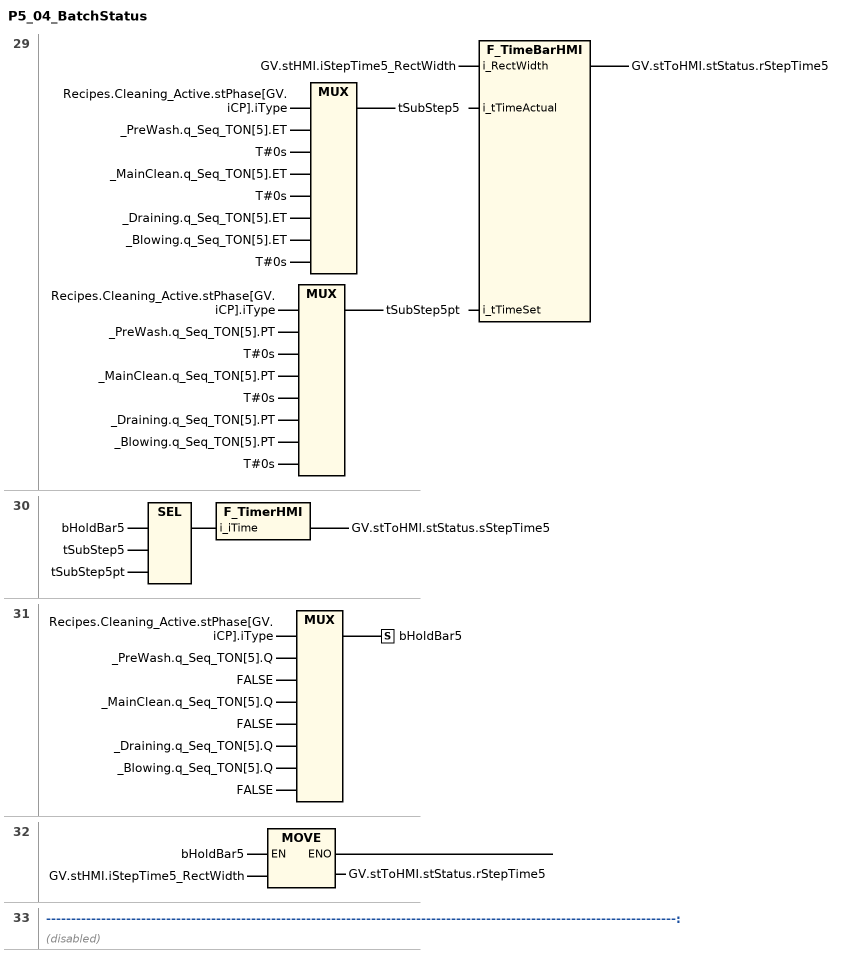
// NETWORK 29
_w10 := MUX(Recipes.Cleaning_Active.stPhase[GV.iCP].iType, _PreWash.q_Seq_TON[5].ET, T#0s, _MainClean.q_Seq_TON[5].ET, T#0s, _Draining.q_Seq_TON[5].ET, _Blowing.q_Seq_TON[5].ET, T#0s);
tSubStep5 := _w10;
_w11 := MUX(Recipes.Cleaning_Active.stPhase[GV.iCP].iType, _PreWash.q_Seq_TON[5].PT, T#0s, _MainClean.q_Seq_TON[5].PT, T#0s, _Draining.q_Seq_TON[5].PT, _Blowing.q_Seq_TON[5].PT, T#0s);
tSubStep5pt := _w11;
GV.stToHMI.stStatus.rStepTime5 := F_TimeBarHMI(i_RectWidth := GV.stHMI.iStepTime5_RectWidth, i_tTimeActual := _w10, i_tTimeSet := _w11);

// NETWORK 30
GV.stToHMI.stStatus.sStepTime5 := F_TimerHMI(i_iTime := SEL(bHoldBar5, tSubStep5, tSubStep5pt));

// NETWORK 31
bHoldBar5 S= MUX(Recipes.Cleaning_Active.stPhase[GV.iCP].iType, _PreWash.q_Seq_TON[5].Q, FALSE, _MainClean.q_Seq_TON[5].Q, FALSE, _Draining.q_Seq_TON[5].Q, _Blowing.q_Seq_TON[5].Q, FALSE);

// NETWORK 32
IF bHoldBar5 THEN GV.stToHMI.stStatus.rStepTime5 := GV.stHMI.iStepTime5_RectWidth; END_IF

// NETWORK 33 (disabled)
// label: ------------------------------------------------------------------------------------------------------------------------------

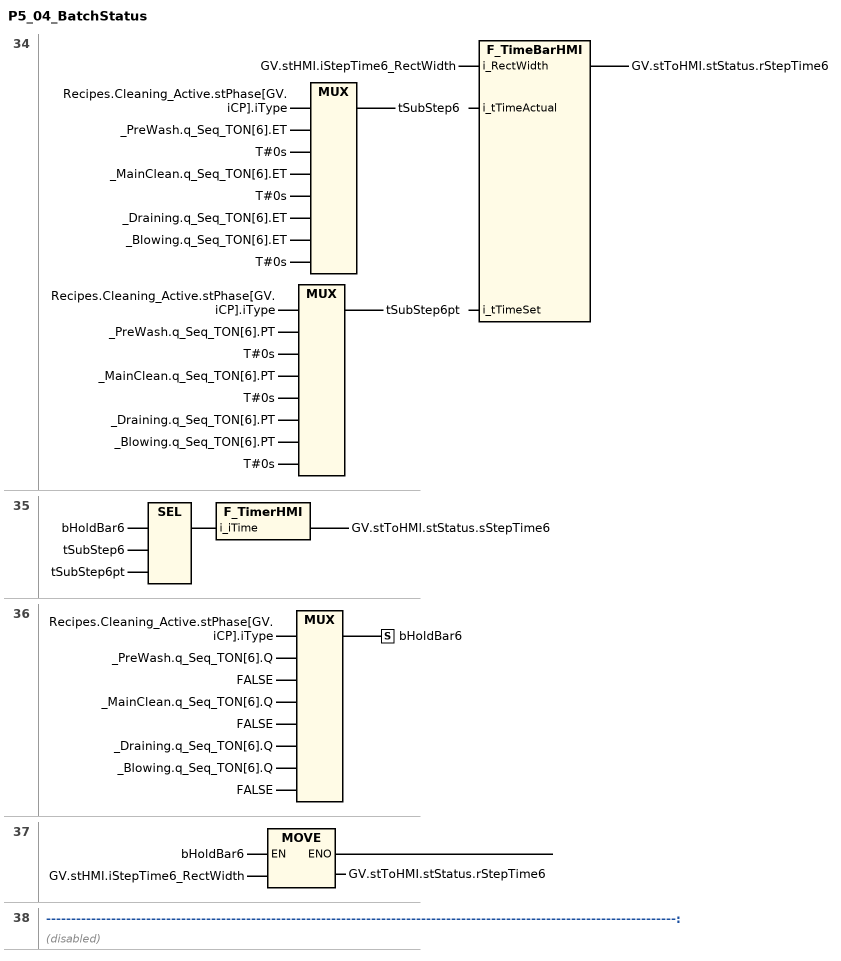
// NETWORK 34
_w12 := MUX(Recipes.Cleaning_Active.stPhase[GV.iCP].iType, _PreWash.q_Seq_TON[6].ET, T#0s, _MainClean.q_Seq_TON[6].ET, T#0s, _Draining.q_Seq_TON[6].ET, _Blowing.q_Seq_TON[6].ET, T#0s);
tSubStep6 := _w12;
_w13 := MUX(Recipes.Cleaning_Active.stPhase[GV.iCP].iType, _PreWash.q_Seq_TON[6].PT, T#0s, _MainClean.q_Seq_TON[6].PT, T#0s, _Draining.q_Seq_TON[6].PT, _Blowing.q_Seq_TON[6].PT, T#0s);
tSubStep6pt := _w13;
GV.stToHMI.stStatus.rStepTime6 := F_TimeBarHMI(i_RectWidth := GV.stHMI.iStepTime6_RectWidth, i_tTimeActual := _w12, i_tTimeSet := _w13);

// NETWORK 35
GV.stToHMI.stStatus.sStepTime6 := F_TimerHMI(i_iTime := SEL(bHoldBar6, tSubStep6, tSubStep6pt));

// NETWORK 36
bHoldBar6 S= MUX(Recipes.Cleaning_Active.stPhase[GV.iCP].iType, _PreWash.q_Seq_TON[6].Q, FALSE, _MainClean.q_Seq_TON[6].Q, FALSE, _Draining.q_Seq_TON[6].Q, _Blowing.q_Seq_TON[6].Q, FALSE);

// NETWORK 37
IF bHoldBar6 THEN GV.stToHMI.stStatus.rStepTime6 := GV.stHMI.iStepTime6_RectWidth; END_IF

// NETWORK 38 (disabled)
// label: ------------------------------------------------------------------------------------------------------------------------------

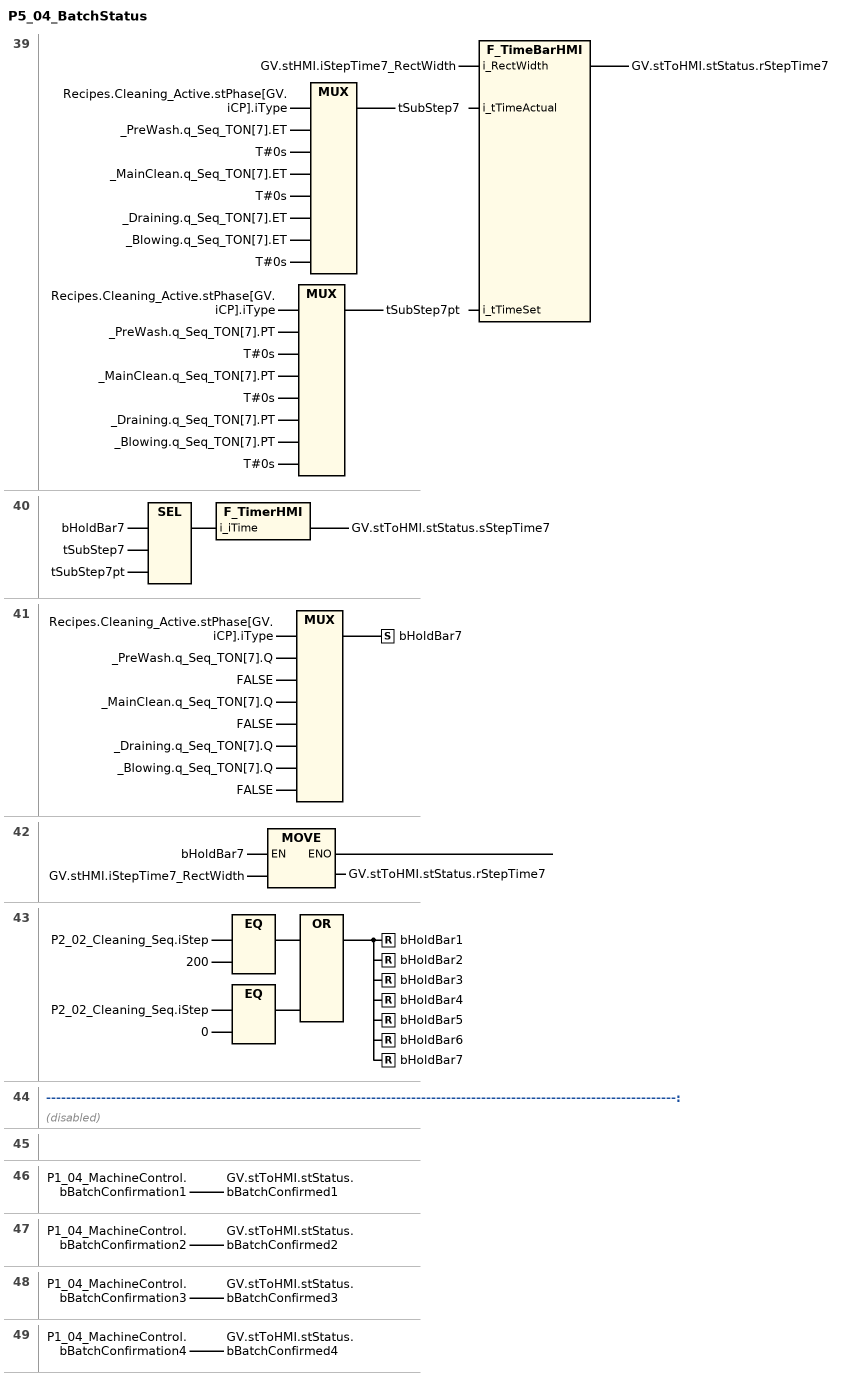
// NETWORK 39
_w14 := MUX(Recipes.Cleaning_Active.stPhase[GV.iCP].iType, _PreWash.q_Seq_TON[7].ET, T#0s, _MainClean.q_Seq_TON[7].ET, T#0s, _Draining.q_Seq_TON[7].ET, _Blowing.q_Seq_TON[7].ET, T#0s);
tSubStep7 := _w14;
_w15 := MUX(Recipes.Cleaning_Active.stPhase[GV.iCP].iType, _PreWash.q_Seq_TON[7].PT, T#0s, _MainClean.q_Seq_TON[7].PT, T#0s, _Draining.q_Seq_TON[7].PT, _Blowing.q_Seq_TON[7].PT, T#0s);
tSubStep7pt := _w15;
GV.stToHMI.stStatus.rStepTime7 := F_TimeBarHMI(i_RectWidth := GV.stHMI.iStepTime7_RectWidth, i_tTimeActual := _w14, i_tTimeSet := _w15);

// NETWORK 40
GV.stToHMI.stStatus.sStepTime7 := F_TimerHMI(i_iTime := SEL(bHoldBar7, tSubStep7, tSubStep7pt));

// NETWORK 41
bHoldBar7 S= MUX(Recipes.Cleaning_Active.stPhase[GV.iCP].iType, _PreWash.q_Seq_TON[7].Q, FALSE, _MainClean.q_Seq_TON[7].Q, FALSE, _Draining.q_Seq_TON[7].Q, _Blowing.q_Seq_TON[7].Q, FALSE);

// NETWORK 42
IF bHoldBar7 THEN GV.stToHMI.stStatus.rStepTime7 := GV.stHMI.iStepTime7_RectWidth; END_IF

// NETWORK 43
_w16 := P2_02_Cleaning_Seq.iStep = 200 OR P2_02_Cleaning_Seq.iStep = 0;
bHoldBar1 R= _w16;
bHoldBar2 R= _w16;
bHoldBar3 R= _w16;
bHoldBar4 R= _w16;
bHoldBar5 R= _w16;
bHoldBar6 R= _w16;
bHoldBar7 R= _w16;

// NETWORK 44 (disabled)
// label: ------------------------------------------------------------------------------------------------------------------------------

// NETWORK 45

// NETWORK 46
GV.stToHMI.stStatus.bBatchConfirmed1 := P1_04_MachineControl.bBatchConfirmation1;

// NETWORK 47
GV.stToHMI.stStatus.bBatchConfirmed2 := P1_04_MachineControl.bBatchConfirmation2;

// NETWORK 48
GV.stToHMI.stStatus.bBatchConfirmed3 := P1_04_MachineControl.bBatchConfirmation3;

// NETWORK 49
GV.stToHMI.stStatus.bBatchConfirmed4 := P1_04_MachineControl.bBatchConfirmation4;

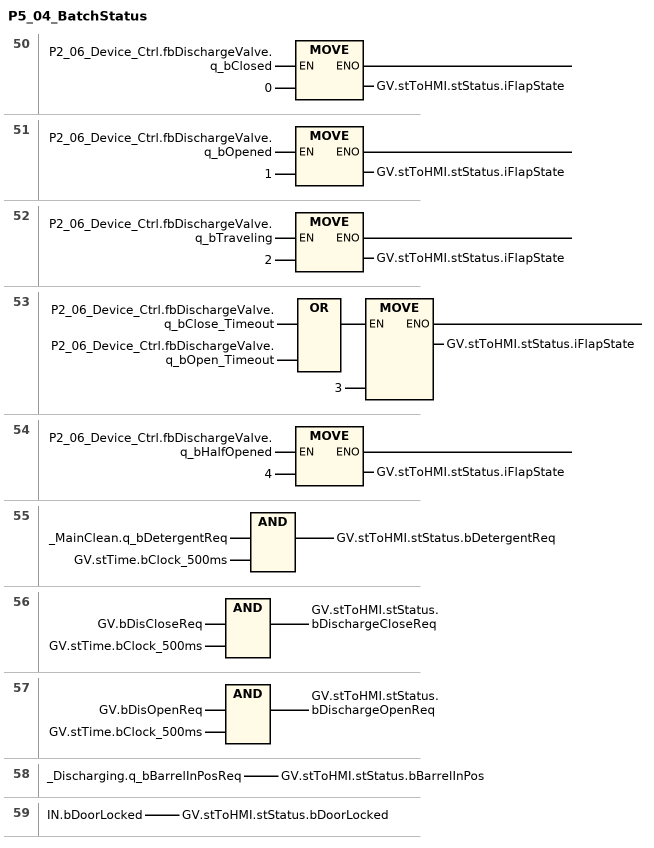
// NETWORK 50
IF P2_06_Device_Ctrl.fbDischargeValve.q_bClosed THEN GV.stToHMI.stStatus.iFlapState := 0; END_IF

// NETWORK 51
IF P2_06_Device_Ctrl.fbDischargeValve.q_bOpened THEN GV.stToHMI.stStatus.iFlapState := 1; END_IF

// NETWORK 52
IF P2_06_Device_Ctrl.fbDischargeValve.q_bTraveling THEN GV.stToHMI.stStatus.iFlapState := 2; END_IF

// NETWORK 53
IF P2_06_Device_Ctrl.fbDischargeValve.q_bClose_Timeout OR P2_06_Device_Ctrl.fbDischargeValve.q_bOpen_Timeout THEN
    GV.stToHMI.stStatus.iFlapState := 3;
END_IF

// NETWORK 54
IF P2_06_Device_Ctrl.fbDischargeValve.q_bHalfOpened THEN GV.stToHMI.stStatus.iFlapState := 4; END_IF

// NETWORK 55
GV.stToHMI.stStatus.bDetergentReq := _MainClean.q_bDetergentReq AND GV.stTime.bClock_500ms;

// NETWORK 56
GV.stToHMI.stStatus.bDischargeCloseReq := GV.bDisCloseReq AND GV.stTime.bClock_500ms;

// NETWORK 57
GV.stToHMI.stStatus.bDischargeOpenReq := GV.bDisOpenReq AND GV.stTime.bClock_500ms;

// NETWORK 58
GV.stToHMI.stStatus.bBarrelInPos := _Discharging.q_bBarrelInPosReq;

// NETWORK 59
GV.stToHMI.stStatus.bDoorLocked := IN.bDoorLocked;

END_PROGRAM

// ---- FB/F_TimerHMI.TcPOU
FUNCTION F_TimerHMI : STRING
VAR_INPUT
	i_iTime				:TIME;
END_VAR
VAR
	iTimeInSec			:UDINT;
	iHours				:UDINT;
	iMinutes			:UDINT;
	iSeconds			:UDINT;
	sQuery				:STRING;
END_VAR

iTimeInSec:=TO_UDINT(i_iTIme)/1000;

iHours:=iTimeInSec/3600;
iMinutes:=(iTimeInSec/60)-(iHours*60);
iSeconds:=iTimeInSec - (iMinutes*60) - (iHours*3600);

IF iHours = 0 THEN
	sQuery:='00:';
ELSIF iHours > 0 AND iHours < 10 THEN
	sQuery:=CONCAT('0',TO_STRING(iHours));
	sQuery:=CONCAT(sQuery,':');
ELSE
	sQuery:=TO_STRING(iHours);
	sQuery:=CONCAT(sQuery,':');
END_IF

IF iMinutes = 0 THEN
	sQuery:=CONCAT(sQuery,'00:');
ELSIF iMinutes > 0 AND iMinutes < 10 THEN
	sQuery:=CONCAT(sQuery,'0');
	sQuery:=CONCAT(sQuery,TO_STRING(iMinutes));
	sQuery:=CONCAT(sQuery,':');
ELSE
	sQuery:=CONCAT(sQuery,TO_STRING(iMinutes));
	sQuery:=CONCAT(sQuery,':');
END_IF

IF iSeconds = 0 THEN
	sQuery:=CONCAT(sQuery,'00');
ELSIF iSeconds > 0 AND iSeconds < 10 THEN
	sQuery:=CONCAT(sQuery,'0');
	sQuery:=CONCAT(sQuery,TO_STRING(iSeconds));
ELSE
	sQuery:=CONCAT(sQuery,TO_STRING(iSeconds));
END_IF


F_TimerHMI:=sQuery;

END_FUNCTION

// ---- FB/F_TimeBarHMI.TcPOU
FUNCTION F_TimeBarHMI : REAL
VAR_INPUT
	i_RectWidth				:INT;
	i_tTimeActual			:TIME;
	i_tTimeSet				:TIME;
END_VAR
VAR
	iTimeActual_Min				:DINT;
	iTimeSet_Min				:DINT;
	fbScale						:FB_Scale;
END_VAR

iTimeSet_Min:=TIME_TO_DINT(i_tTimeSet)/100;
iTimeActual_Min:=TIME_TO_DINT(i_tTimeActual)/100;

IF iTimeSet_Min <> 0 THEN
	fbSCale(i_rValue:=DINT_TO_REAL(iTimeActual_Min),
			i_rRawData_Low:=0,
			i_rRawData_High:=DINT_TO_INT(iTimeSet_Min),
			i_rScaled_Low:=0,
			i_rScaled_High:=i_RectWidth,
			i_rOffset:=0,
			q_rScaled=>F_TimeBarHMI);
END_IF

END_FUNCTION

// ---- POUs/5. HMI/P5_05_Screenshot.TcPOU
PROGRAM P5_05_Screenshot
VAR
		fbScreenshot					:NT_StartProcess;
		tonDisable						:TON;
		bDisable						:BOOL;
END_VAR

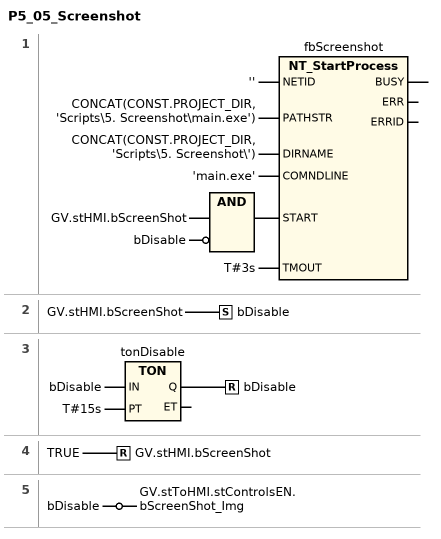
// NETWORK 1
fbScreenshot(
    NETID := '',
    PATHSTR := CONCAT(CONST.PROJECT_DIR,'Scripts\5. Screenshot\main.exe'),
    DIRNAME := CONCAT(CONST.PROJECT_DIR,'Scripts\5. Screenshot\'),
    COMNDLINE := 'main.exe',
    START := GV.stHMI.bScreenShot AND NOT bDisable,
    TMOUT := T#3s); // NT_StartProcess

// NETWORK 2
bDisable S= GV.stHMI.bScreenShot;

// NETWORK 3
tonDisable(IN := bDisable, PT := T#15s); // TON
bDisable R= tonDisable.Q;

// NETWORK 4
GV.stHMI.bScreenShot R= TRUE;

// NETWORK 5
GV.stToHMI.stControlsEN.bScreenShot_Img := NOT bDisable;

END_PROGRAM

// ---- POUs/5. HMI/P5_06_Trends.TcPOU
PROGRAM P5_06_Trends
VAR
END_VAR

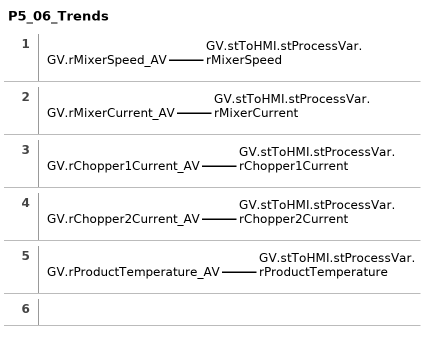
// NETWORK 1
GV.stToHMI.stProcessVar.rMixerSpeed := GV.rMixerSpeed_AV;

// NETWORK 2
GV.stToHMI.stProcessVar.rMixerCurrent := GV.rMixerCurrent_AV;

// NETWORK 3
GV.stToHMI.stProcessVar.rChopper1Current := GV.rChopper1Current_AV;

// NETWORK 4
GV.stToHMI.stProcessVar.rChopper2Current := GV.rChopper2Current_AV;

// NETWORK 5
GV.stToHMI.stProcessVar.rProductTemperature := GV.rProductTemperature_AV;

// NETWORK 6

END_PROGRAM

// ---- FB/Database/FB_WriteEvent.TcPOU
FUNCTION_BLOCK FB_WriteEvent
VAR_INPUT
	i_bWrite		:BOOL;
	i_enEvent		:EN_BatchEvents;
	i_sDescription	:STRING;
END_VAR
VAR
	Trig			:R_TRIG;
END_VAR
VAR_IN_OUT
	iq_stParams		:ST_OperatorAct;
	iq_bWrite		:BOOL;
END_VAR

Trig(CLK:=i_bWrite);
IF Trig.Q THEN
	iq_stParams.Event:=TO_STRING(i_enEvent);
	iq_stParams.Description := i_sDescription;
	iq_bWrite:=TRUE;
END_IF

END_FUNCTION_BLOCK

// ---- FB/FB_Coil_Ctrl.TcPOU
FUNCTION_BLOCK FB_Coil_Ctrl
VAR_INPUT
	i_Interlocks		:ARRAY[1..5] OF BOOL;
	i_AutoCmd			:BOOL;
	i_ManCmd			:BOOL;
	i_ServiceMode		:BOOL;
END_VAR
VAR_OUTPUT
	q_InterlocksOK		:BOOL;
	q_bCmd				:BOOL;
END_VAR
VAR
	bCmd				:BOOL;
	tofCMD				:TOF;
END_VAR

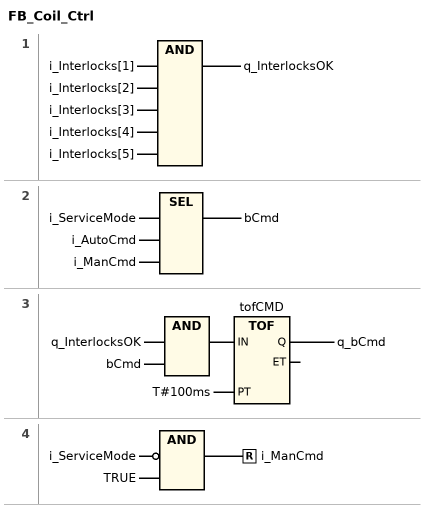
// NETWORK 1
q_InterlocksOK := i_Interlocks[1] AND i_Interlocks[2] AND i_Interlocks[3] AND i_Interlocks[4] AND i_Interlocks[5];

// NETWORK 2
bCmd := SEL(i_ServiceMode, i_AutoCmd, i_ManCmd);

// NETWORK 3
tofCMD(IN := q_InterlocksOK AND bCmd, PT := T#100ms); // TOF
q_bCmd := tofCMD.Q;

// NETWORK 4
i_ManCmd R= NOT i_ServiceMode AND TRUE;

END_FUNCTION_BLOCK

// ---- FB/FB_FileSaveAs_V02.TcPOU
FUNCTION_BLOCK FB_FileSaveAs_V02
VAR_INPUT
	i_bExecute					:BOOL;
	i_sSourcePath				:STRING;
	i_sDestinationPath			:STRING;
	i_sFileSourceName			:STRING;
	i_sFileDestName				:STRING;
END_VAR
VAR_OUTPUT
	q_bBusy						:BOOL;
	q_bDone						:BOOL;
	q_bError					:BOOL;
	q_sError					:STRING;
END_VAR
VAR
	fbSourceOpen				:FB_FileOpen;
	fbDestinationOpen			:FB_FileOpen;
	
	fbSourceRead				:FB_FileRead;
	fbDestinationWrite			:FB_FileWrite;
	
	fbSourceClose				:FB_FileClose;
	fbDestinationClose			:FB_FileClose;
	
	sSourceOpen					:STRING[300];
	sDestinationOpen			:STRING[300];

	arrData						:ARRAY[0..9999] OF BYTE;
	
	bOpen						:BOOL;
	bRead						:BOOL;
	bWrite						:BOOL;
	bClose						:BOOL;
	
	iStep						:INT;
END_VAR


CASE iStep OF
	
	0:
		q_bBusy:=FALSE;
		IF i_bExecute THEN
			q_sError:='';
			q_bError:=FALSE;
			q_bDone:=FALSE;
			q_bBusy:=TRUE;
			MEMSET(ADR(arrData),0,SIZEOF(arrData));
			iStep:=10;
		END_IF

	10:
		sSourceOpen := CONCAT(i_sSourcePath,i_sFileSourceName);
		sDestinationOpen := CONCAT(i_sDestinationPath,i_sFileDestName);
		iStep:=20;
		
	20:
		bOpen:=TRUE;
		IF NOT fbSourceOpen.bBusy AND NOT fbDestinationOpen.bBusy AND NOT fbSourceOpen.bError AND NOT fbDestinationOpen.bError THEN
			iStep:=30;
		ELSIF fbSourceOpen.bError OR fbDestinationOpen.bError THEN
			q_bError:=TRUE;
			q_sError:='Error opening files';
			iStep:=50;
		END_IF
		
	30:
		bRead:=TRUE;
		IF fbSourceRead.bBusy THEN
			iStep:=35;
		END_IF
	35:
		
		IF NOT fbSourceRead.bBusy AND NOT fbSourceRead.bError THEN
			iStep:=40;
		ELSIF fbSourceRead.bError THEN
			q_bError:=TRUE;
			q_sError:='Error reading source file';
			iStep:=50;
		END_IF
		
	40:
		bWrite:=TRUE;
		IF fbDestinationWrite.bBusy THEN
			iStep:=45;
		END_IF
	45:
		IF NOT fbDestinationWrite.bBusy AND NOT fbDestinationWrite.bError THEN
			iStep:=50;
		ELSIF fbDestinationWrite.bError THEN
			q_bError:=TRUE;
			q_sError:='Error writing source file';
			iStep:=50;
		END_IF
	50:
		bClose:=TRUE;
		IF NOT fbSourceClose.bBusy AND NOT fbDestinationClose.bBusy AND NOT fbSourceClose.bError AND NOT fbDestinationClose.bError THEN
			iStep:=100;
		ELSIF fbSourceClose.bError OR fbDestinationClose.bError THEN
			q_bError:=TRUE;
			q_sError:='Error closing files';
			iStep:=0;
		END_IF
		
	100:
		q_bDone:=TRUE;
		iStep:=0;
	
END_CASE

Cmd();

ACTION Cmd:
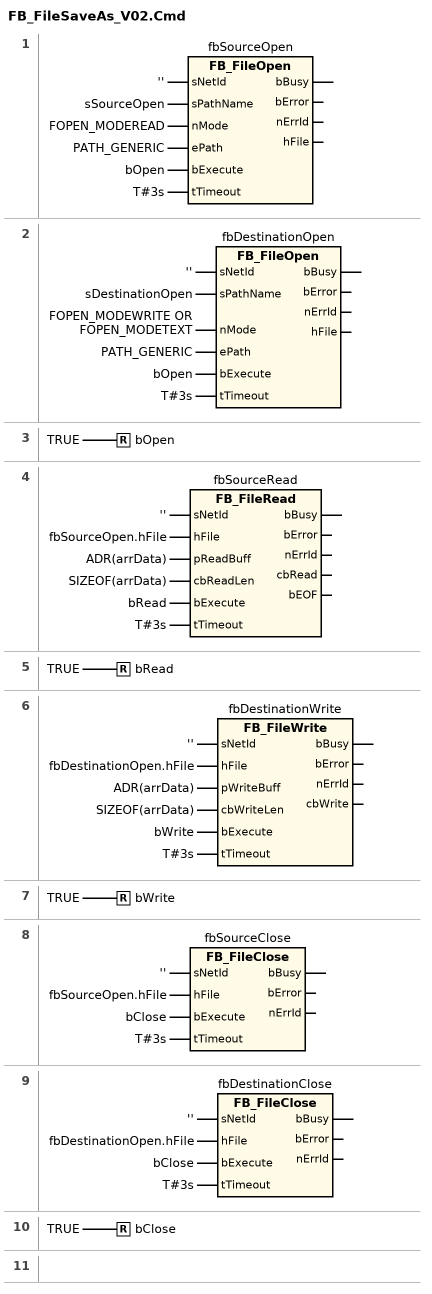
// NETWORK 1
fbSourceOpen(
    sNetId := '',
    sPathName := sSourceOpen,
    nMode := FOPEN_MODEREAD,
    ePath := PATH_GENERIC,
    bExecute := bOpen,
    tTimeout := T#3s); // FB_FileOpen

// NETWORK 2
fbDestinationOpen(
    sNetId := '',
    sPathName := sDestinationOpen,
    nMode := FOPEN_MODEWRITE OR FOPEN_MODETEXT,
    ePath := PATH_GENERIC,
    bExecute := bOpen,
    tTimeout := T#3s); // FB_FileOpen

// NETWORK 3
bOpen R= TRUE;

// NETWORK 4
fbSourceRead(
    sNetId := '',
    hFile := fbSourceOpen.hFile,
    pReadBuff := ADR(arrData),
    cbReadLen := SIZEOF(arrData),
    bExecute := bRead,
    tTimeout := T#3s); // FB_FileRead

// NETWORK 5
bRead R= TRUE;

// NETWORK 6
fbDestinationWrite(
    sNetId := '',
    hFile := fbDestinationOpen.hFile,
    pWriteBuff := ADR(arrData),
    cbWriteLen := SIZEOF(arrData),
    bExecute := bWrite,
    tTimeout := T#3s); // FB_FileWrite

// NETWORK 7
bWrite R= TRUE;

// NETWORK 8
fbSourceClose(sNetId := '', hFile := fbSourceOpen.hFile, bExecute := bClose, tTimeout := T#3s); // FB_FileClose

// NETWORK 9
fbDestinationClose(sNetId := '', hFile := fbDestinationOpen.hFile, bExecute := bClose, tTimeout := T#3s); // FB_FileClose

// NETWORK 10
bClose R= TRUE;

// NETWORK 11
END_ACTION

END_FUNCTION_BLOCK

// ---- FB/FB_TimeElapsed_HMI.TcPOU
FUNCTION_BLOCK FB_TimeElapsed_HMI
VAR_INPUT
	i_RectWidth				:INT;
	i_tTimeActual			:TIME;
	i_tTimeSet				:TIME;
END_VAR
VAR_OUTPUT
	q_iValue				:REAL;
END_VAR
VAR
	iTimeActual_Min				:DINT;
	iTimeSet_Min				:DINT;
	fbScale						:FB_Scale;
END_VAR

iTimeSet_Min:=TIME_TO_DINT(i_tTimeSet)/100;
iTimeActual_Min:=TIME_TO_DINT(i_tTimeActual)/100;

IF iTimeSet_Min <> 0 THEN
	fbSCale(i_iValue:=DINT_TO_INT(iTimeActual_Min),
			i_iRawData_Low:=0,
			i_iRawData_High:=DINT_TO_INT(iTimeSet_Min),
			i_rScaled_Low:=0,
			i_rScaled_High:=i_RectWidth,
			i_rOffset:=0,
			q_rScaled=>q_iValue);
END_IF

END_FUNCTION_BLOCK

// ---- FB/F_OperationalTime.TcPOU
FUNCTION F_OperationalTime : ARRAY[0..2] OF INT
VAR_INPUT
	i_min				:UDINT;
END_VAR
VAR
	dayMins				:INT;
	hourMins			:INT;
	day					:INT;
	hour				:INT;
	mins				:INT;
END_VAR

day:=TO_INT(i_min/(60*24));
dayMins:=day*60*24;
hour:=TO_INT(i_min-TO_UDINT(dayMins))/60;
hourMins:=hour*60;
mins:=TO_INT(i_min-TO_UDINT(dayMins))-hourMins;

F_OperationalTime[0]:=day;
F_OperationalTime[1]:=hour;
F_OperationalTime[2]:=mins;

END_FUNCTION
